Universal Robots PolyScope program: ricardonicolasP1.urp

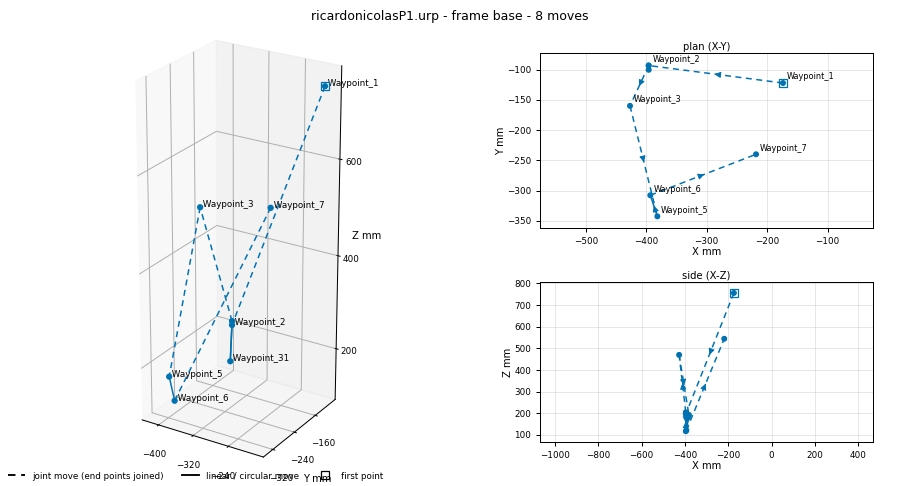
[picture p0: tool path of ricardonicolasP1.urp in frame base, 8 of 8 moves have a stored position in this frame; points joined in program order, loops and branches not executed]
Program ricardonicolasP1 (installation=ricardoNicolasP1 directory=/programs createdIn=5.9.3.1031212 lastSavedIn=5.9.3.1031212 robotSerialNumber=20195300809)
Calibrated DH parameters: a=[-0.000085, -0.20076, -0.212369, 0.000121, -0.000118, 0]; d=[0.15185, -26.306375, 24.753047, 1.684739, 0.085386, 0.092088]; alpha=[1.572149, -0.00522, -0.011864, 1.571339, -1.571085, 0]; deltaTheta=[0, 0.599885, -0.513355, -0.086555, 0.000006, 0]
InitVariablesNode variables(variable(name=PiezaHome, expression=False))
Robot Program (runOnlyOnce=false)
  Wait DigitalInput pin=digital_in[0]; digitalValue=1
  URCap Gripper (Robotiq_Grippers, Robotiq Inc.) dataModel(position=0.0, force=0.0, speed=100.0, positionInDouble=0.0, forceInDouble=0.0, speedInDouble=100.0, slaveIds=[9], blocking=true)
  MoveJ speed 60 deg/s, acceleration 80 deg/s^2 (useActiveTCP=true) feature=Base
    Waypoint Waypoint_1: TCP in base x=-173.872 y=-122.21 z=756.214 mm, rx=-0.8584 ry=-0.9065 rz=1.2406 rad; joints [-3.025, -122.317, 50.377, -131.795, -90.731, -6.675] deg; TCP offset x=0 y=0 z=200 mm, rx=0 ry=0 rz=0 rad
    Waypoint Waypoint_2: TCP in base x=-396.012 y=-93.326 z=196.137 mm, rx=-2.0996 ry=-2.2238 rz=0.04 rad; joints [-4.3, -67.56, 39.021, -66.099, -92.659, -7.328] deg; TCP offset x=0 y=0 z=200 mm, rx=0 ry=0 rz=0 rad
  MoveL speed 250 mm/s, acceleration 1200 mm/s^2 (useActiveTCP=true) feature=Base
    Waypoint Waypoint_31: TCP in base x=-395.867 y=-100.356 z=117.543 mm, rx=-2.0995 ry=-2.2239 rz=0.04 rad; joints [-3.211, -73.58, 69.625, -90.659, -92.763, -6.506] deg
  URCap Gripper (Robotiq_Grippers, Robotiq Inc.) dataModel(position=100.0, force=0.0, speed=100.0, positionInDouble=100.0, forceInDouble=0.0, speedInDouble=100.0, slaveIds=[9], blocking=true)
  MoveL speed 250 mm/s, acceleration 1200 mm/s^2 (useActiveTCP=true) feature=Base
    Waypoint Waypoint_4: TCP in base x=-396.002 y=-93.301 z=204.896 mm, rx=-2.0997 ry=-2.2238 rz=0.0398 rad; joints [-4.295, -65.748, 33.515, -62.397, -92.65, -7.288] deg
  MoveJ speed 60 deg/s, acceleration 80 deg/s^2 (useActiveTCP=true) feature=Base
    Waypoint Waypoint_3: TCP in base x=-426.827 y=-159.959 z=470.071 mm, rx=-1.8769 ry=-1.611 rz=1.0258 rad; joints [-2.123, -77.447, 12.566, -76.571, -82.193, 10.897] deg
    Waypoint Waypoint_5: TCP in base x=-381.597 y=-342.674 z=192.752 mm, rx=-2.0478 ry=-2.1977 rz=0.3441 rad; joints [28.423, -41.5, 0.751, -63.799, -93.092, 24.29] deg
  MoveL speed 250 mm/s, acceleration 1200 mm/s^2 (useActiveTCP=true) feature=Base
    Waypoint Waypoint_6: TCP in base x=-393.261 y=-307.795 z=121.554 mm, rx=-2.0888 ry=-2.1568 rz=0.1271 rad; joints [26.23, -47.025, 28.575, -78.771, -96.614, 24.116] deg
  URCap Gripper (Robotiq_Grippers, Robotiq Inc.) dataModel(position=0.0, force=0.0, speed=100.0, positionInDouble=0.0, forceInDouble=0.0, speedInDouble=100.0, slaveIds=[9], blocking=true)
  MoveJ speed 60 deg/s, acceleration 80 deg/s^2 (useActiveTCP=true) feature=Base
    Waypoint Waypoint_7: TCP in base x=-218.439 y=-240.018 z=544.511 mm, rx=-1.6967 ry=-1.712 rz=1.3315 rad; joints [27.606, -90.272, 3.227, -64.491, -94.821, 25.004] deg
  Wait Sleep waitTime=1
  PiezaHome := True
Thread Thread_1 (runOnlyOnce=false)
  Set AnalogOutput pin=analog_out[1]; analogValue=4
  Set AnalogOutput pin=analog_out[0]; analogValue=3
  Wait DigitalInput pin=digital_in[0]; digitalValue=1
  Set AnalogOutput pin=analog_out[1]; analogValue=0
  Wait Condition expression=PiezaHome≟ True
  Script: sync()
